# EPICS substitutions: siteApps-725b29e158e8061764313f5708af9e46fe30c0a8/siteApps-725b29e158e8061764313f5708af9e46fe30c0a8/Tr1/tr1App/Db/user.substitutions
# Example substitutions file

file "db/dbExample1.db" {
    { user = "root" }
}

file db/dbExample2.db {
    pattern { user, no, scan }
        { "root", 1, "1 second" }
        { "root", 2, "2 second" }
        { "root", 3, "5 second" }
}
